Update(
    stDataSource:=stSourceDataStore[3],
    sName:='LS3 (From laser bay 2)',
    fbSourceValve:=GVL_BTS_VAC.fb_LS3_VGC,
    fbLinear:=GVL_BTPS.fbLS3Linear,
    fbRotary:=GVL_BTPS.fbLS3Rotary,
    fbGoniometer:=GVL_BTPS.fbLS3Goniometer,
    fbNearField:=GVL_BTPS.fbLS3NearFieldCamStats,
    fbFarField:=GVL_BTPS.fbLS3FarFieldCamStats
);

Update(
    stDataSource:=stSourceDataStore[4],
    sName:='LS4 (From laser bay 2)',
    fbSourceValve:=GVL_BTS_VAC.fb_LS4_VGC,
    fbLinear:=GVL_BTPS.fbLS4Linear,
    fbRotary:=GVL_BTPS.fbLS4Rotary,
    fbGoniometer:=GVL_BTPS.fbLS4Goniometer,
    fbNearField:=GVL_BTPS.fbLS4NearFieldCamStats,
    fbFarField:=GVL_BTPS.fbLS4FarFieldCamStats
);

Update(
    stDataSource:=stSourceDataStore[6],
    sName:='LS6 (From laser bay 3)',
    fbSourceValve:=GVL_BTS_VAC.fb_LS6_VGC,
    fbLinear:=GVL_BTPS.fbLS6Linear,
    fbRotary:=GVL_BTPS.fbLS6Rotary,
    fbGoniometer:=GVL_BTPS.fbLS6Goniometer,
    fbNearField:=GVL_BTPS.fbLS6NearFieldCamStats,
    fbFarField:=GVL_BTPS.fbLS6FarFieldCamStats
);

METHOD Update : BOOL
VAR_INPUT
    sName : STRING;
END_VAR
VAR_IN_OUT
    // The data source to update
    stDataSource : ST_SourceDataStore;

    // The source information
    fbSourceValve : FB_VGC;
    fbNearField : FB_EpicsStatsMonitor;
    fbFarField : FB_EpicsStatsMonitor;
    fbLinear : FB_EpicsMotorMonitor;
    fbRotary : FB_EpicsMotorMonitor;
    fbGoniometer : FB_EpicsMotorMonitor;

END_VAR
stDataSource.sName := sName;
stDataSource.fbSourceValve REF= fbSourceValve;

stDataSource.bEntryValveReady := F_IsValveReady(fbSourceValve);

(* Update range comparisons with their source values *)
(* Cameras *)
stDataSource.fbNFCentroidX.fValue := fbNearField.fCentroidX;
stDataSource.fbNFCentroidX.bInputValid := fbNearField.bValid AND fbNearField.bIsUpdating;
stDataSource.fbNFCentroidY.fValue := fbNearField.fCentroidY;
stDataSource.fbNFCentroidY.bInputValid := fbNearField.bValid AND fbNearField.bIsUpdating;
stDataSource.fbFFCentroidX.fValue := fbFarField.fCentroidX;
stDataSource.fbFFCentroidX.bInputValid := fbFarField.bValid AND fbFarField.bIsUpdating;
stDataSource.fbFFCentroidY.fValue := fbFarField.fCentroidY;
stDataSource.fbFFCentroidY.bInputValid := fbFarField.bValid AND fbFarField.bIsUpdating;

(* Motors *)
stDataSource.fbLinear.fValue := fbLinear.fPosition;
stDataSource.fbLinear.bInputValid := fbLinear.bValid AND fbLinear.stMSTA.bHomed (* AND fbLinear.stMSTA.bClosedLoop *);
stDataSource.fbRotary.fValue := fbRotary.fPosition;
stDataSource.fbRotary.bInputValid := fbRotary.bValid AND fbRotary.stMSTA.bHomed (* AND fbRotary.stMSTA.bClosedLoop *);
stDataSource.fbGoniometer.fValue := fbGoniometer.fPosition;
stDataSource.fbGoniometer.bInputValid := fbGoniometer.bValid AND fbGoniometer.stMSTA.bHomed (* AND fbGoniometer.stMSTA.bClosedLoop *);

(* Run the range comparisons *)
stDataSource.fbNFCentroidX();
stDataSource.fbNFCentroidY();
stDataSource.fbFFCentroidX();
stDataSource.fbFFCentroidY();
stDataSource.fbLinear();
stDataSource.fbRotary();
stDataSource.fbGoniometer();

(* Data is valid overall if *all* range comparisons say so *)
stDataSource.bDataValid := (
    stDataSource.fbNFCentroidX.bInputValid AND
    stDataSource.fbNFCentroidY.bInputValid AND
    stDataSource.fbFFCentroidX.bInputValid AND
    stDataSource.fbFFCentroidY.bInputValid AND
    stDataSource.fbLinear.bInputValid AND
    stDataSource.fbRotary.bInputValid AND
    stDataSource.fbGoniometer.bInputValid AND
    TRUE
);

(* Checks only pass if data is valid and all comparisons are true *)
stDataSource.bChecksOK := (
    stDataSource.bDataValid AND
    stDataSource.fbNFCentroidX.bInRange AND
    stDataSource.fbNFCentroidY.bInRange AND
    stDataSource.fbFFCentroidX.bInRange AND
    stDataSource.fbFFCentroidY.bInRange AND
    stDataSource.fbLinear.bInRange AND
    stDataSource.fbRotary.bInRange AND
    stDataSource.fbGoniometer.bInRange AND
    stDataSource.bEntryValveReady AND
    bExitValveReady AND
    TRUE
);

stDataSource.bInPosition := stDataSource.fbLinear.bInputValid AND stDataSource.fbLinear.bInRange;
END_METHOD

END_FUNCTION_BLOCK

// ---- POUs/BTPS/FB_RangeComparison.TcPOU
FUNCTION_BLOCK FB_RangeComparison
VAR_INPUT PERSISTENT
    (* The low part of the range. *)
    {attribute 'pytmc' := 'pv: Low'}
    fLow : LREAL;
    (* The high part of the range. *)
    {attribute 'pytmc' := 'pv: High'}
    fHigh : LREAL;
    (* Nominal value for this.  User-facing value. *)
    {attribute 'pytmc' := '
        pv: Nominal
        io: io
        field: DESC Nominal value for setting
    '}
    fNominal : LREAL;
    (* Are the limits inclusive? *)
    {attribute 'pytmc' := '
        pv: Inclusive
        field: ZNAM Exclusive
        field: ONAM Inclusive
    '}
    bInclusive : BOOL := TRUE;
END_VAR
VAR_INPUT
    (* The input value for comparison *)
    {attribute 'pytmc' := 'pv: Value; io: input'}
    fValue : LREAL;
    (* Should the input value be trusted? *)
    {attribute 'pytmc' := '
        pv: Valid
        io: input
        field: ZNAM Data Invalid
        field: ONAM Data Valid
        field: ZSV MAJOR
        field: OSV NO_ALARM
    '}
    bInputValid : BOOL := FALSE;

END_VAR
VAR_OUTPUT
    {attribute 'pytmc' := '
        pv: InRange
        io: input
        field: ZNAM Out of range
        field: ONAM In range
        field: ZSV MAJOR
        field: OSV NO_ALARM
    '}
    bInRange : BOOL;
END_VAR

IF NOT bInputValid OR fHigh < fLow THEN
    bInRange := FALSE;
ELSIF bInclusive THEN
    bInRange := (fValue >= fLow) AND (fValue <= fHigh);
ELSE
    bInRange := (fValue > fLow) AND (fValue < fHigh);
END_IF

END_FUNCTION_BLOCK

// ---- POUs/BTPS/Tests/FB_TestRangeComparison.TcPOU
{attribute 'call_after_init'}
FUNCTION_BLOCK FB_TestRangeComparison EXTENDS TcUnit.FB_TestSuite
VAR_INPUT
END_VAR
VAR_OUTPUT
END_VAR
VAR
    fbRange : FB_RangeComparison;
END_VAR

TEST('Inclusive valid data');

fbRange.fLow := 0.0;
fbRange.fHigh := 10.0;
fbRange.fNominal := 0.0;
fbRange.bInclusive := TRUE;
fbRange.bInputValid := TRUE;

fbRange(fValue:=0.0);
AssertTrue(fbRange.bInRange, Message:='lower bound');
fbRange(fValue:=10.0);
AssertTrue(fbRange.bInRange, Message:='upper bound');
fbRange(fValue:=5.0);
AssertTrue(fbRange.bInRange, Message:='mid range');
fbRange(fValue:=-1.0);
AssertFalse(fbRange.bInRange, Message:='below range');
fbRange(fValue:=11.0);
AssertFalse(fbRange.bInRange, Message:='above range');

TEST_FINISHED();

TEST('Exclusive valid data');

fbRange.fLow := 0.0;
fbRange.fHigh := 10.0;
fbRange.fNominal := 0.0;
fbRange.bInclusive := FALSE;
fbRange.bInputValid := TRUE;

fbRange(fValue:=0.0);
AssertFalse(fbRange.bInRange, Message:='lower bound');
fbRange(fValue:=10.0);
AssertFalse(fbRange.bInRange, Message:='upper bound');
fbRange(fValue:=5.0);
AssertTrue(fbRange.bInRange, Message:='mid range');
fbRange(fValue:=-1.0);
AssertFalse(fbRange.bInRange, Message:='below range');
fbRange(fValue:=11.0);
AssertFalse(fbRange.bInRange, Message:='above range');

TEST_FINISHED();

TEST('Invalid data');

fbRange.fLow := 0.0;
fbRange.fHigh := 10.0;
fbRange.fNominal := 0.0;
fbRange.bInclusive := TRUE;
fbRange.bInputValid := FALSE;

fbRange(fValue:=0.0);
AssertFalse(fbRange.bInRange, Message:='lower bound');
fbRange(fValue:=10.0);
AssertFalse(fbRange.bInRange, Message:='upper bound');
fbRange(fValue:=5.0);
AssertFalse(fbRange.bInRange, Message:='mid range');
fbRange(fValue:=-1.0);
AssertFalse(fbRange.bInRange, Message:='below range');
fbRange(fValue:=11.0);
AssertFalse(fbRange.bInRange, Message:='above range');

TEST_FINISHED();


TEST('Bad range');

fbRange.fLow := 0.0;
fbRange.fHigh := 0.0;
fbRange.fNominal := 0.0;
fbRange.bInclusive := TRUE;
fbRange.bInputValid := FALSE;

fbRange(fValue:=0.0);
AssertFalse(fbRange.bInRange, Message:='lower bound');
fbRange(fValue:=10.0);
AssertFalse(fbRange.bInRange, Message:='upper bound');
fbRange(fValue:=5.0);
AssertFalse(fbRange.bInRange, Message:='mid range');
fbRange(fValue:=-1.0);
AssertFalse(fbRange.bInRange, Message:='below range');
fbRange(fValue:=11.0);
AssertFalse(fbRange.bInRange, Message:='above range');

TEST_FINISHED();

END_FUNCTION_BLOCK

// ---- POUs/BTPS/Tests/FB_TestShutterSafety.TcPOU
FUNCTION_BLOCK FB_TestShutterSafety EXTENDS TcUnit.FB_TestSuite
VAR_INPUT
END_VAR
VAR_OUTPUT
END_VAR
VAR
    fbShutter : FB_ShutterSafety;
    fbDestinations : ARRAY [1..GVL_BTPS_Constants.nDestinations] OF FB_DestinationDataStore;
    nDest : UINT;
    nSource : UINT;
END_VAR

TEST('Bad source index');

Reset();

fbShutter.bAcknowledge := FALSE;
fbShutter.bUserOpenRequest := FALSE;
fbShutter.bOverride := FALSE;
fbShutter.nSourceIndex := 0;

fbShutter(fbDestinations:=fbDestinations);
AssertFalse(fbShutter.bSafeToOpen, Message:='Bad source index');

TEST_FINISHED();

TEST('Safe to open');

Reset();

fbDestinations[1].stSourceDataStore[1].bChecksOK := TRUE;

fbShutter.bAcknowledge := FALSE;
fbShutter.bOverride := FALSE;

fbShutter(nSourceIndex:=1, bUserOpenRequest:=FALSE, fbDestinations:=fbDestinations);
AssertTrue(fbShutter.bSafeToOpen, Message:='Safe for source 1');
AssertFalse(fbShutter.bOpenSignal, Message:='Safe for source 1; close');
fbShutter(nSourceIndex:=1, bUserOpenRequest:=TRUE, fbDestinations:=fbDestinations);
AssertTrue(fbShutter.bSafeToOpen, Message:='Safe for source 1');
AssertTrue(fbShutter.bOpenSignal, Message:='Safe for source 1; open');

fbShutter(nSourceIndex:=2, bUserOpenRequest:=TRUE, fbDestinations:=fbDestinations);
AssertFalse(fbShutter.bSafeToOpen, Message:='Not safe for source 2');
AssertFalse(fbShutter.bOpenSignal, Message:='Not safe for source 2; close');

TEST_FINISHED();



TEST('Acknowledge error');

Reset();

fbDestinations[1].stSourceDataStore[1].bChecksOK := FALSE;
fbShutter(nSourceIndex:=1, bUserOpenRequest:=TRUE, fbDestinations:=fbDestinations, bAcknowledge:=False);
AssertFalse(fbShutter.bSafeToOpen, Message:='Not safe yet');
AssertFalse(fbShutter.bOpenSignal, Message:='Not safe yet; close');
AssertFalse(fbShutter.bUserOpenRequest, Message:='Reset open request on fail');
AssertTrue(fbShutter.bLatchedError, Message:='Latched error');

fbDestinations[1].stSourceDataStore[1].bChecksOK := TRUE;
fbShutter(nSourceIndex:=1, fbDestinations:=fbDestinations, bAcknowledge:=TRUE);
AssertTrue(fbShutter.bSafeToOpen, Message:='Safe for source 2');
AssertFalse(fbShutter.bOpenSignal, Message:='Open not yet requested');
AssertFalse(fbShutter.bLatchedError, Message:='Latched error cleared');

fbShutter(nSourceIndex:=1, bUserOpenRequest:=TRUE, fbDestinations:=fbDestinations, bAcknowledge:=FALSE);
AssertTrue(fbShutter.bSafeToOpen, Message:='Safe for source 2');
AssertTrue(fbShutter.bOpenSignal, Message:='Safe for source 2; open');
AssertFalse(fbShutter.bLatchedError, Message:='Latched error cleared');

TEST_FINISHED();



TEST('Override error');

Reset();

fbDestinations[1].stSourceDataStore[1].bChecksOK := FALSE;
fbShutter(nSourceIndex:=1, bUserOpenRequest:=TRUE, fbDestinations:=fbDestinations, bAcknowledge:=False);
AssertFalse(fbShutter.bSafeToOpen, Message:='Not safe yet');
AssertFalse(fbShutter.bOpenSignal, Message:='Not safe yet; close');
AssertFalse(fbShutter.bUserOpenRequest, Message:='Reset open request on fail');
AssertTrue(fbShutter.bLatchedError, Message:='Latched error');

fbShutter.bOverride := TRUE;

fbShutter(nSourceIndex:=1, fbDestinations:=fbDestinations);
AssertTrue(fbShutter.bSafeToOpen, Message:='Safe for source 2');
AssertFalse(fbShutter.bOpenSignal, Message:='Open not yet requested');
AssertTrue(fbShutter.bLatchedError, Message:='Latched error overridden not cleared');

fbShutter(nSourceIndex:=1, bUserOpenRequest:=TRUE, fbDestinations:=fbDestinations);
AssertTrue(fbShutter.bSafeToOpen, Message:='Safe for source 2');
AssertTrue(fbShutter.bOpenSignal, Message:='Safe for source 2; open');
AssertFalse(fbShutter.bLatchedError, Message:='Latched error still there');

fbShutter(nSourceIndex:=1, bUserOpenRequest:=FALSE, fbDestinations:=fbDestinations);
AssertTrue(fbShutter.bSafeToOpen, Message:='Safe for source 2');
AssertTrue(fbShutter.bOpenSignal, Message:='Safe for source 2; open');
AssertFalse(fbShutter.bLatchedError, Message:='Latched error still there');
AssertFalse(fbShutter.bOverride, Message:='Override set after shutter closure');

TEST_FINISHED();

ACTION Reset:
fbShutter.bAcknowledge := TRUE;
fbShutter.bUserOpenRequest := FALSE;
fbShutter.bOverride := TRUE;
fbShutter.nSourceIndex := 1;

fbShutter(fbDestinations:=fbDestinations);

fbShutter.bAcknowledge := FALSE;
fbShutter.bUserOpenRequest := FALSE;
fbShutter.bOverride := FALSE;
fbShutter.nSourceIndex := 1;

fbShutter(fbDestinations:=fbDestinations);

FOR nDest := 1 TO GVL_BTPS_Constants.nDestinations DO
    fbDestinations[nDest].stSourceDataStore[nSource].bChecksOK := FALSE;
END_FOR

WRITE_PROTECTED_BOOL(ADR(fbShutter.bLatchedError), FALSE);
WRITE_PROTECTED_BOOL(ADR(fbShutter.bOpenSignal), FALSE);
WRITE_PROTECTED_BOOL(ADR(fbShutter.bSafeToOpen), FALSE);
END_ACTION

END_FUNCTION_BLOCK

// ---- POUs/BTPS/Tests/FB_Test_EpicsCentroidMonitor.TcPOU
{attribute 'call_after_init'}
FUNCTION_BLOCK FB_Test_EpicsCentroidMonitor EXTENDS TcUnit.FB_TestSuite
VAR_INPUT
END_VAR
VAR_OUTPUT
END_VAR
VAR
END_VAR

TestBasics();

METHOD TestBasics
VAR_INPUT
END_VAR
VAR_INST
    fbMonitor : FB_EpicsStatsMonitor;
    nCount : INT := 0;
END_VAR
TEST('Updating_OK');

fbMonitor.nMaxDroppedFrames := 2;
fbMonitor.fMaximumFrameTime := 10.0;
fbMonitor.fMinPixelSumChange := 0.5;

WriteCentroidValue(fbMonitor:=fbMonitor, tLastUpdate:=T#0S, fX:=0.0, fY:=0.0, fTotal:=0.0, nCount:=nCount, nX_Severity:=0, nY_Severity:=0, nCount_Severity:=0, nTotal_Severity:=0);
fbMonitor();

WriteCentroidValue(fbMonitor:=fbMonitor, tLastUpdate:=T#1S, fX:=0.1, fY:=0.1, fTotal:=1.0, nCount:=nCount, nX_Severity:=0, nY_Severity:=0, nCount_Severity:=0, nTotal_Severity:=0);
fbMonitor();

WriteCentroidValue(fbMonitor:=fbMonitor, tLastUpdate:=T#2S, fX:=0.1, fY:=0.1, fTotal:=2.0, nCount:=nCount, nX_Severity:=0, nY_Severity:=0, nCount_Severity:=0, nTotal_Severity:=0);
fbMonitor();

AssertTrue(fbMonitor.bIsUpdating, Message:='Centroid not reporting updating');
AssertEquals_LREAL(fbMonitor.fFrameTime, 1.5, 1E-6, Message:='Update time inaccurate');
AssertEquals_LREAL(fbMonitor.fFrameTimes[1], 1.0, 1E-6, Message:='Update time inaccurate');
AssertEquals_LREAL(fbMonitor.fFrameTimes[2], 2.0, 1E-6, Message:='Update time inaccurate');

WriteCentroidValue(fbMonitor:=fbMonitor, tLastUpdate:=T#2S, fX:=0.1, fY:=0.1, fTotal:=3.0, nCount:=nCount, nX_Severity:=0, nY_Severity:=0, nCount_Severity:=0, nTotal_Severity:=0);
fbMonitor();

AssertEquals_LREAL(fbMonitor.fFrameTimes[1], 2.0, 1E-6, Message:='Update time inaccurate');
AssertEquals_LREAL(fbMonitor.fFrameTimes[2], 2.0, 1E-6, Message:='Update time inaccurate');

TEST_FINISHED();

(*
TEST('Updating_Not_OK');

fbMonitor.Initialize();

fbMonitor.nMaxDroppedFrames := 2;
fbMonitor.fMaximumFrameTime := 10.0;
fbMonitor.fMinPixelSumChange := 0.5;

WriteCentroidValue(fbMonitor:=fbMonitor, tLastUpdate:=T#0S, fX:=0.0, fY:=0.0, fTotal:=0.0, nCount:=nCount, nX_Severity:=0, nY_Severity:=0, nCount_Severity:=0, nTotal_Severity:=0);
fbMonitor();

WriteCentroidValue(fbMonitor:=fbMonitor, tLastUpdate:=T#11S, fX:=0.1, fY:=0.1, fTotal:=0.0, nCount:=nCount, nX_Severity:=0, nY_Severity:=0, nCount_Severity:=0, nTotal_Severity:=0);
fbMonitor();

WriteCentroidValue(fbMonitor:=fbMonitor, tLastUpdate:=T#11S, fX:=0.1, fY:=0.1, fTotal:=0.0, nCount:=nCount, nX_Severity:=0, nY_Severity:=0, nCount_Severity:=0, nTotal_Severity:=0);
fbMonitor();

AssertFalse(fbMonitor.bIsUpdating, Message:='Centroid not updating');
AssertEquals_LREAL(fbMonitor.fFrameTime, fbMonitor.fMaximumFrameTime, 1E-6, Message:='Update time inaccurate');
AssertEquals_LREAL(fbMonitor.fFrameTimes[1], fbMonitor.fMaximumFrameTime, 1E-6, Message:='Update time inaccurate');
AssertEquals_LREAL(fbMonitor.fFrameTimes[2], fbMonitor.fMaximumFrameTime, 1E-6, Message:='Update time inaccurate');

TEST_FINISHED();

// TODO: how to make that timer trigger?
*)

TEST('Severity invalidation');

WriteCentroidValue(fbMonitor:=fbMonitor, fX:=0.0, fY:=0.0, fTotal:=0.0, nCount:=nCount, nX_Severity:=2, nY_Severity:=0, nCount_Severity:=0, nTotal_Severity:=0, tLastUpdate:=T#0.2S);
fbMonitor(fMinPixelSumChange:=0.0);
AssertFalse(fbMonitor.bValid, Message:='Invalid data - x severity');

WriteCentroidValue(fbMonitor:=fbMonitor, fX:=0.1, fY:=0.1, fTotal:=0.0, nCount:=nCount, nX_Severity:=0, nY_Severity:=2, nCount_Severity:=0, nTotal_Severity:=0, tLastUpdate:=T#0.2S);
fbMonitor(fMinPixelSumChange:=0.0);
AssertFalse(fbMonitor.bValid, Message:='Invalid data - y severity');

WriteCentroidValue(fbMonitor:=fbMonitor, fX:=0.2, fY:=0.2, fTotal:=0.0, nCount:=nCount, nX_Severity:=0, nY_Severity:=0, nCount_Severity:=2, nTotal_Severity:=0, tLastUpdate:=T#0.2S);
fbMonitor(fMinPixelSumChange:=0.0);
AssertFalse(fbMonitor.bValid, Message:='Invalid data - count severity');

WriteCentroidValue(fbMonitor:=fbMonitor, fX:=0.2, fY:=0.2, fTotal:=0.0, nCount:=nCount, nX_Severity:=0, nY_Severity:=0, nCount_Severity:=0, nTotal_Severity:=2, tLastUpdate:=T#0.2S);
fbMonitor(fMinPixelSumChange:=0.0);
AssertFalse(fbMonitor.bValid, Message:='Invalid data - total severity');

WriteCentroidValue(fbMonitor:=fbMonitor, fX:=0.0, fY:=0.0, fTotal:=fbMonitor.fMinPixelSumChange, nCount:=nCount, nX_Severity:=0, nY_Severity:=0, nCount_Severity:=0, nTotal_Severity:=0, tLastUpdate:=T#0.1S);
fbMonitor(fMinPixelSumChange:=0.0);
AssertTrue(fbMonitor.bValid, Message:='Data valid');
AssertTrue(fbMonitor.bIsUpdating, Message:='Data valid and updating');

TEST_FINISHED();
END_METHOD

METHOD WriteCentroidValue
VAR_IN_OUT
    fbMonitor : FB_EpicsStatsMonitor;
END_VAR
VAR_INPUT
    fX : LREAL;
    fY : LREAL;
    fTotal : LREAL;
    nCount : INT;
    nX_Severity : INT := 0;
    nY_Severity : INT := 0;
    nCount_Severity : INT := 0;
    nTotal_Severity : INT := 0;
    tLastUpdate : TIME;
END_VAR
WRITE_PROTECTED_INT(ADR(fbMonitor.fbCentroidX.iPLCInternalSeverity), nX_Severity);
WRITE_PROTECTED_INT(ADR(fbMonitor.fbCentroidY.iPLCInternalSeverity), nY_Severity);
WRITE_PROTECTED_INT(ADR(fbMonitor.fbArrayCounter.iPLCInternalSeverity), nCount_Severity);
WRITE_PROTECTED_INT(ADR(fbMonitor.fbTotal.iPLCInternalSeverity), nTotal_Severity);

WRITE_PROTECTED_LREAL(ADR(fbMonitor.fbCentroidX.fPLCInternalValue), fX);
WRITE_PROTECTED_LREAL(ADR(fbMonitor.fbCentroidY.fPLCInternalValue), fY);
WRITE_PROTECTED_LREAL(ADR(fbMonitor.fbTotal.fPLCInternalValue), fTotal);
WRITE_PROTECTED_LREAL(ADR(fbMonitor.fbArrayCounter.fPLCInternalValue), INT_TO_LREAL(nCount));

WRITE_PROTECTED_TIME(ADR(fbMonitor.tLastUpdate), TIME() - tLastUpdate);
END_METHOD

END_FUNCTION_BLOCK

// ---- POUs/BTPS/Tests/PRG_RunTests.TcPOU
PROGRAM PRG_RunTests
VAR
    fbRangeComparison : FB_TestRangeComparison;
    fbShutterSafety : FB_TestShutterSafety;
    fbCentroidTest : FB_Test_EpicsCentroidMonitor;
    fbMotorTest : FB_Test_EpicsMotorMonitor;

END_VAR

TcUnit.RUN();

END_PROGRAM
